TYPE ST_Error :
STRUCT
	Error			: BOOL := FALSE;
	Reason			: STRING := '';
END_STRUCT
END_TYPE

(* stored: Version 1.1.0.1, ProductVersion 3.1.4026.18
   DUT ST_Error: Id {eab08672-e8c6-4020-94d1-f51b24dde733} *)
